(* PLC project Untitled1, Beckhoff Automation GmbH TwinCAT PLC Control 3.5.13.21 *)
(* stored: creationDateTime 2024-10-30T15:48:25.8174981, modificationDateTime 2024-10-30T15:48:25.8201123 *)

FUNCTION_BLOCK FB_EdgeDetector
VAR_INPUT
	inputValue : BOOL;
	DoublePressedTime: UINT;
END_VAR
VAR_OUTPUT
	risingEdge : BOOL;
	fallingEdge : BOOL;
	DoublePressed: BOOL;
END_VAR
VAR
	inputValue_old : BOOL;
	OncePressed: BOOL := FALSE;
	DoublePressedcounter: UINT := 0;
END_VAR

            risingEdge := FALSE;
fallingEdge := FALSE;
DoublePressed := FALSE;

IF inputValue <> inputValue_old THEN
	IF inputValue = TRUE THEN
		risingEdge := TRUE;
		IF OncePressed = FALSE THEN
			OncePressed := TRUE;
		ELSE
			OncePressed := FALSE;
			DoublePressed := TRUE;
			DoublePressedcounter := 0;
		END_IF
	ELSE
		fallingEdge := TRUE;
	END_IF
END_IF
inputValue_old := inputValue;
IF OncePressed = TRUE THEN
	IF DoublePressedcounter >= DoublePressedTime THEN
		OncePressed := FALSE;
		DoublePressedcounter := 0;
	ELSE
		DoublePressedcounter := DoublePressedcounter + 1;
	END_IF	
END_IF

          
END_FUNCTION_BLOCK
